// Implicitly generated code : DO NOT EDIT
FUNCTION CheckDivDInt : DINT
VAR_INPUT
	divisor:DINT;
END_VAR

// Implicitly generated code : Only an Implementation suggestion
IF divisor = 0 THEN
	CheckDivDInt:=1;
	GVL_Checks.dCheckDivDInt := GVL_Checks.dCheckDivDInt + 1;
ELSE
	CheckDivDInt:=divisor;
END_IF;

END_FUNCTION

(* stored: Version 1.1.0.1, ProductVersion 3.1.4020.3
   POU CheckDivDInt: Id {503361d9-0c2e-4512-8202-4d7e24803e7c}, SpecialFunc CheckDivInt32 *)
